FUNCTION IsGreaterthanten : BOOL
VAR_INPUT
	rValue : INT;
END_VAR
VAR
END_VAR

IF rValue>10 THEN
	IsGreaterthanten := TRUE;
END_IF

END_FUNCTION

(* stored: Version 1.1.0.1, ProductVersion 3.1.4024.16
   POU IsGreaterthanten: Id {08b81fda-5b4c-4061-9a58-4e2fe8a8e7ad}, SpecialFunc None *)
